// TIA Portal V18 export
FUNCTION_BLOCK "CMMS_Z1_Movement"   // FB14, LAD
{ S7_Optimized_Access := 'TRUE' }
VERSION : 0.1
// stored: AutoNumber true, IsIECCheckEnabled false, IsRetainMemResEnabled false, MemoryReserve 100, SetENOAutomatically false, UDAEnableTagReadback false
   VAR
      FML_REF { S7_SetPoint := 'True'} : "DT_FML_REF";
   END_VAR
   // FML_REF.DeviceType := 'CMMS';
BEGIN

REGION Network 1
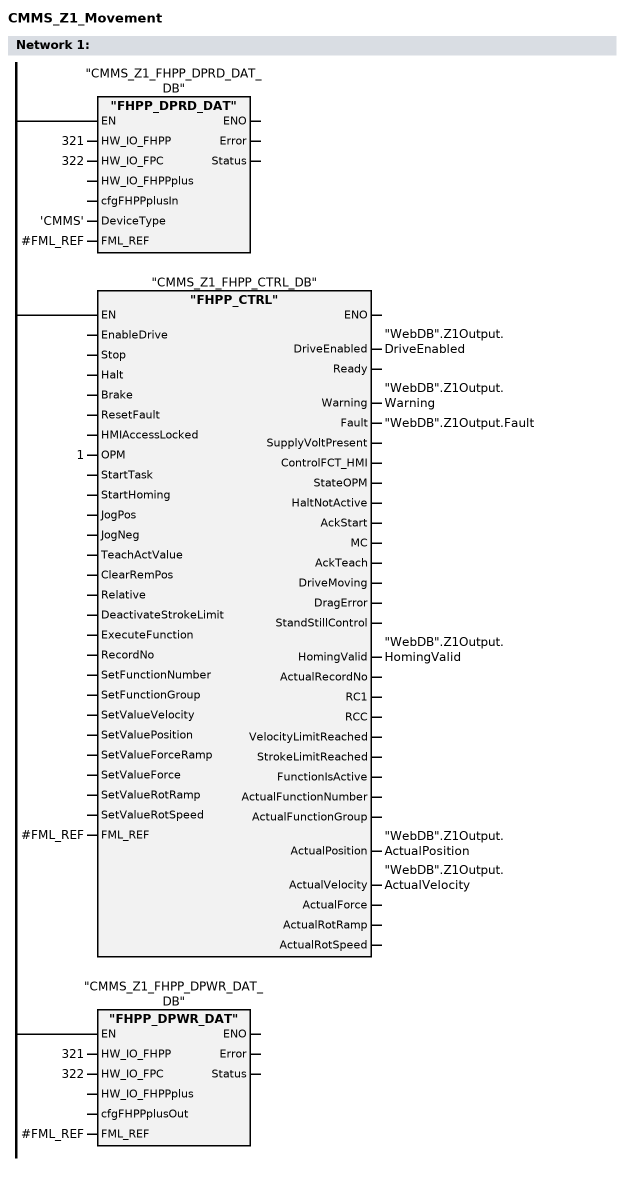
   RUNG wire#powerrail
      "CMMS_Z1_FHPP_DPRD_DAT_DB"(HW_IO_FHPP := 321, HW_IO_FPC := 322, HW_IO_FHPPplus :=, cfgFHPPplusIn :=, DeviceType := 'CMMS', FML_REF := #FML_REF, Error =>, Status =>)
   END_RUNG
   RUNG wire#powerrail
      "CMMS_Z1_FHPP_CTRL_DB"(EnableDrive :=, Stop :=, Halt :=, Brake :=, ResetFault :=, HMIAccessLocked :=, OPM := 1, StartTask :=, StartHoming :=, JogPos :=, JogNeg :=, TeachActValue :=, ClearRemPos :=, Relative :=, DeactivateStrokeLimit :=, ExecuteFunction :=, RecordNo :=, SetFunctionNumber :=, SetFunctionGroup :=, SetValueVelocity :=, SetValuePosition :=, SetValueForceRamp :=, SetValueForce :=, SetValueRotRamp :=, SetValueRotSpeed :=, FML_REF := #FML_REF, DriveEnabled => "WebDB".Z1Output.DriveEnabled, Ready =>, Warning => "WebDB".Z1Output.Warning, Fault => "WebDB".Z1Output.Fault, SupplyVoltPresent =>, ControlFCT_HMI =>, StateOPM =>, HaltNotActive =>, AckStart =>, MC =>, AckTeach =>, DriveMoving =>, DragError =>, StandStillControl =>, HomingValid => "WebDB".Z1Output.HomingValid, ActualRecordNo =>, RC1 =>, RCC =>, VelocityLimitReached =>, StrokeLimitReached =>, FunctionIsActive =>, ActualFunctionNumber =>, ActualFunctionGroup =>, ActualPosition => "WebDB".Z1Output.ActualPosition, ActualVelocity => "WebDB".Z1Output.ActualVelocity, ActualForce =>, ActualRotRamp =>, ActualRotSpeed =>)
   END_RUNG
   RUNG wire#powerrail
      "CMMS_Z1_FHPP_DPWR_DAT_DB"(HW_IO_FHPP := 321, HW_IO_FPC := 322, HW_IO_FHPPplus :=, cfgFHPPplusOut :=, FML_REF := #FML_REF, Error =>, Status =>)
   END_RUNG
   // the same network as SCL:
   "CMMS_Z1_FHPP_DPRD_DAT_DB"(HW_IO_FHPP := 321, HW_IO_FPC := 322, DeviceType := 'CMMS', FML_REF := #FML_REF);   // "FHPP_DPRD_DAT"
   "CMMS_Z1_FHPP_CTRL_DB"(OPM := 1,   // "FHPP_CTRL"
                          FML_REF := #FML_REF,
                          DriveEnabled => "WebDB".Z1Output.DriveEnabled,
                          Warning => "WebDB".Z1Output.Warning,
                          Fault => "WebDB".Z1Output.Fault,
                          HomingValid => "WebDB".Z1Output.HomingValid,
                          ActualPosition => "WebDB".Z1Output.ActualPosition,
                          ActualVelocity => "WebDB".Z1Output.ActualVelocity);
   "CMMS_Z1_FHPP_DPWR_DAT_DB"(HW_IO_FHPP := 321, HW_IO_FPC := 322, FML_REF := #FML_REF);   // "FHPP_DPWR_DAT"
END_REGION
END_FUNCTION_BLOCK
